FUNCTION_BLOCK FB_Module01 EXTENDS FB_ModuleBase
VAR_INPUT
END_VAR
VAR_OUTPUT
END_VAR
VAR
	fbComponent1:				FB_Component;
	fbComponent2:				FB_Component;
	fbComponent3:				FB_ComponentEx;
END_VAR

METHOD PUBLIC M_Cycle
VAR_INPUT
END_VAR
SUPER^.M_Cycle();

fbComponent1.M_Cycle();
fbComponent2.M_Cycle();
fbComponent3.M_Cycle();
END_METHOD

METHOD PROTECTED M_Execute : bool
VAR_INPUT
END_VAR
M_Execute:= SUPER^.M_Execute() AND FALSE;

IF bWarning THEN
	fbEvent.M_Warning('My secound Warning', '' );	
END_IF
END_METHOD

METHOD PROTECTED M_Initialise
VAR_INPUT
END_VAR
SUPER^.M_Initialise();

P_ID:= '1';

M_Attach(fbComponent1);
M_Attach(fbComponent2);
M_Attach(fbComponent3);
END_METHOD

METHOD PROTECTED M_Running
VAR_INPUT
END_VAR
//IF NOT M001.fbEmStop.P_Value THEN
//	fbEvent.M_AddSTRING(M001.fbEmStop.P_ID);
//	fbEvent.M_Abort('Emergency stop not ok', '');
//ELSIF NOT M001.fbPowerOn.P_Value THEN
//	fbEvent.M_AddSTRING(M001.fbPowerOn.P_ID);
//	fbEvent.M_Abort('Power not on', '');
//ELSIF NOT M001.fbFuse1.P_Value THEN
//	fbEvent.M_AddSTRING(M001.fbFuse1.P_ID);
//	fbEvent.M_Stop('Fuse Triped', '');	
	
//END_IF
END_METHOD

METHOD PROTECTED M_Starting : BOOL
VAR_INPUT
END_VAR
M_Starting:= SUPER^.M_Starting();
END_METHOD

METHOD PROTECTED M_Stopping : BOOL // Return state complete
VAR_INPUT
END_VAR
// State Stopping
M_Stopping:= SUPER^.M_Stopping();
END_METHOD

END_FUNCTION_BLOCK

(* stored: Version 1.1.0.1, ProductVersion 3.1.4024.12
   POU FB_Module01: Id {3744d03d-359c-4ab8-84fb-4ea93b7a5162}, SpecialFunc None
   Method M_Cycle: Id {655447dc-389e-494a-be91-78d8a111b7aa}
   Method M_Execute: Id {0f7f4331-8af5-0744-015a-f65d0021dd06}
   Method M_Initialise: Id {714c485c-83a6-4af2-a706-fec3f6b598e5}
   Method M_Running: Id {eaffebca-5ff2-4f17-be84-3310a9ace22e}
   Method M_Starting: Id {6f002794-61fc-043c-1d84-a8bc502c5d3a}
   Method M_Stopping: Id {478c517c-d184-0eaf-2697-597088f6cf3f} *)
